{attribute 'global_init_slot' := '40510'}
VAR_GLOBAL
  LblFun_Requirement                                       :FB_BA_Label:=( sObjName:='REQ', sDescr:='Requirement');
  LblFun_SystemSwitch                                      :FB_BA_Label:=( sObjName:='PLS', sDescr:='Plant switch');
  LblFun_StatusOccupiedRoom                                :FB_BA_Label:=( sObjName:='OCC', sDescr:='Occupied status room');
  LblFun_LimitCalculatedValue                              :FB_BA_Label:=( sObjName:='LMC', sDescr:='Calculated limit value');
  LblFun_SetpointCalculated                                :FB_BA_Label:=( sObjName:='SPC', sDescr:='Calculated setpoint');
  LblFun_ReadyForOperation                                 :FB_BA_Label:=( sObjName:='RFO', sDescr:='Ready for operation');
  LblFun_OperationalMessage                                :FB_BA_Label:=( sObjName:='OM_', sDescr:='Operational message');
  LblFun_HoursOfOperation                                  :FB_BA_Label:=( sObjName:='OH_', sDescr:='Operating hours');
  LblFun_LimitValueHoursOfOperation                        :FB_BA_Label:=( sObjName:='OHL', sDescr:='Operating hours limit value');
  LblFun_ObjectCalendar                                    :FB_BA_Label:=( sObjName:='CAL', sDescr:='Calendar object');
  LblFun_ObjectCommand                                     :FB_BA_Label:=( sObjName:='COM', sDescr:='Command object');
  LblFun_DifferentialConstantController                    :FB_BA_Label:=( sObjName:='TV_', sDescr:='Differential constant controller');
  LblFun_SwitchOnErrorUnauthorisedON                       :FB_BA_Label:=( sObjName:='SWE', sDescr:='Switch-on error, unauthorised ON');
  LblFun_EnergyLevel                                       :FB_BA_Label:=( sObjName:='EL_', sDescr:='Energy level');
  LblFun_EnergyLevelCalculated                             :FB_BA_Label:=( sObjName:='ELC', sDescr:='Energy level calculated');
  LblFun_UnlockingDevice                                   :FB_BA_Label:=( sObjName:='UNL', sDescr:='Unlocking device');
  LblFun_ObjectEventEnrollment                             :FB_BA_Label:=( sObjName:='EE_', sDescr:='Event enrollment object');
  LblFun_Enabled                                           :FB_BA_Label:=( sObjName:='EN_', sDescr:='Enabled');
  LblFun_DangerAlarm                                       :FB_BA_Label:=( sObjName:='DA_', sDescr:='Danger alarm');
  LblFun_Threshold                                         :FB_BA_Label:=( sObjName:='LM_', sDescr:='Limit value');
  LblFun_LimitMAX                                          :FB_BA_Label:=( sObjName:='LMX', sDescr:='MAX limit');
  LblFun_LimitMIN                                          :FB_BA_Label:=( sObjName:='LMI', sDescr:='MIN limit');
  LblFun_LimitNight                                        :FB_BA_Label:=( sObjName:='LMN', sDescr:='Night limit');
  LblFun_LimitDay                                          :FB_BA_Label:=( sObjName:='LMD', sDescr:='Day limit');
  LblFun_ObjectGroup                                       :FB_BA_Label:=( sObjName:='GP_', sDescr:='Group object');
  LblFun_localPriorityAndOperatingUnitsManualMessage       :FB_BA_Label:=( sObjName:='MNM', sDescr:='local priority and operating units manual message');
  LblFun_HeatingCharacteristicCurveExponent                :FB_BA_Label:=( sObjName:='HEX', sDescr:='Heating characteristic curve exponent');
  LblFun_HeatingCharacteristicCurveParallelDisplacement    :FB_BA_Label:=( sObjName:='HPD', sDescr:='Heating characteristic curve parallel displacement');
  LblFun_HeatingCharacteristicCurveSteepness               :FB_BA_Label:=( sObjName:='HST', sDescr:='Heating characteristic curve steepness');
  LblFun_HeatingCircuitNightReduction                      :FB_BA_Label:=( sObjName:='NGT', sDescr:='Heating circuit night reduction');
  LblFun_Hysteresis                                        :FB_BA_Label:=( sObjName:='HYS', sDescr:='Hysteresis');
  LblFun_Calendar                                          :FB_BA_Label:=( sObjName:='CAL', sDescr:='Calendar');
  LblFun_RuntimeError                                      :FB_BA_Label:=( sObjName:='RUN', sDescr:='Runtime error');
  LblFun_LoopMAXLimit                                      :FB_BA_Label:=( sObjName:='LPX', sDescr:='Loop MAX limit');
  LblFun_LoopMINLimit                                      :FB_BA_Label:=( sObjName:='LPI', sDescr:='Loop MIN limit');
  LblFun_LoopObject                                        :FB_BA_Label:=( sObjName:='LP_', sDescr:='Loop object (controller object) – complex object');
  LblFun_LoopObjectCascadeSupplyAirTemperature             :FB_BA_Label:=( sObjName:='LP_', sDescr:='Cascade controller supply air temperature ');
  LblFun_LoopObjectCascadeSupplyAirHumidity                :FB_BA_Label:=( sObjName:='LP_', sDescr:='Cascade controller supply air humidity ');
  LblFun_MaximumValue                                      :FB_BA_Label:=( sObjName:='MAX', sDescr:='Maximum value');
  LblFun_MeasuredValue                                     :FB_BA_Label:=( sObjName:='MV_', sDescr:='Measured value');
  LblFun_MeasuredValueCalculated                           :FB_BA_Label:=( sObjName:='MVC', sDescr:='Measured value calculated');
  LblFun_MeasuredValueEast                                 :FB_BA_Label:=( sObjName:='MV_', sDescr:='Measured value East');
  LblFun_MeasuredValueNorth                                :FB_BA_Label:=( sObjName:='MV_', sDescr:='Measured value North');
  LblFun_MeasuredValueSouth                                :FB_BA_Label:=( sObjName:='MV_', sDescr:='Measured value South');
  LblFun_MeasuredValueWest                                 :FB_BA_Label:=( sObjName:='MV_', sDescr:='Measured value West');
  LblFun_MinimumValue                                      :FB_BA_Label:=( sObjName:='MIN', sDescr:='Minimum value');
  LblFun_Mean                                              :FB_BA_Label:=( sObjName:='MVL', sDescr:='Mean value');
  LblFun_FollowUpTime                                      :FB_BA_Label:=( sObjName:='FUT', sDescr:='Follow-up time');
  LblFun_ResetTime                                         :FB_BA_Label:=( sObjName:='RST', sDescr:='Reset time');
  LblFun_FeedbackDelay                                     :FB_BA_Label:=( sObjName:='TDF', sDescr:='Time delay feedback');
  LblFun_ObjectNotificationClass                           :FB_BA_Label:=( sObjName:='NC_', sDescr:='Notification class object');
  LblFun_EventClassObject                                  :FB_BA_Label:=( sObjName:='ECL', sDescr:='Event class');
  LblFun_Programobject                                     :FB_BA_Label:=( sObjName:='PRG', sDescr:='Program');
  LblFun_ProportionalBand                                  :FB_BA_Label:=( sObjName:='XP_', sDescr:='Proportional band');
  LblFun_FeedbackOPEN                                      :FB_BA_Label:=( sObjName:='FDO', sDescr:='Feedback OPEN');
  LblFun_FeedbackCLOSED                                    :FB_BA_Label:=( sObjName:='FDC', sDescr:='Feedback CLOSED');
  LblFun_FeedbackValue                                     :FB_BA_Label:=( sObjName:='FDB', sDescr:='Feedback value');
  LblFun_FeedbackErrorOPEN                                 :FB_BA_Label:=( sObjName:='FEO', sDescr:='Feedback error OPEN');
  LblFun_FeedbackErrorCLOSED                               :FB_BA_Label:=( sObjName:='FEC', sDescr:='Feedback error CLOSED');
  LblFun_Feedback                                          :FB_BA_Label:=( sObjName:='FDB', sDescr:='Feedback');
  LblFun_ExecutionControl                                  :FB_BA_Label:=( sObjName:='EXC', sDescr:='Execution control');
  LblFun_SwitchingCommand                                  :FB_BA_Label:=( sObjName:='SC_', sDescr:='Switching command');
  LblFun_Scheduler                                         :FB_BA_Label:=( sObjName:='SCH', sDescr:='Scheduler');
  LblFun_Setpoint                                          :FB_BA_Label:=( sObjName:='SP_', sDescr:='Setpoint');
  LblFun_SetpointComfortHeating                            :FB_BA_Label:=( sObjName:='SP_', sDescr:='Setpoint comfort heating');
  LblFun_SetpointPreComfortHeating                         :FB_BA_Label:=( sObjName:='SP_', sDescr:='Setpoint pre-comfort heating');
  LblFun_SetpointEconomyHeating                            :FB_BA_Label:=( sObjName:='SP_', sDescr:='Setpoint economy heating');
  LblFun_SetpointProtectionHeating                         :FB_BA_Label:=( sObjName:='SP_', sDescr:='Setpoint protection heating');
  LblFun_SetpointComfortCooling                            :FB_BA_Label:=( sObjName:='SP_', sDescr:='Setpoint comfort cooling');
  LblFun_SetpointPreComfortCooling                         :FB_BA_Label:=( sObjName:='SP_', sDescr:='Setpoint pre-comfort cooling');
  LblFun_SetpointEconomyCooling                            :FB_BA_Label:=( sObjName:='SP_', sDescr:='Setpoint economy cooling');
  LblFun_SetpointProtectionCooling                         :FB_BA_Label:=( sObjName:='SP_', sDescr:='Setpoint protection cooling');
  LblFun_SetpointBase                                      :FB_BA_Label:=( sObjName:='SPB', sDescr:='Base setpoint');
  LblFun_SetpointHeating                                   :FB_BA_Label:=( sObjName:='SPH', sDescr:='Heating setpoint');
  LblFun_SetpointCooling                                   :FB_BA_Label:=( sObjName:='SPC', sDescr:='Cooling setpoint');
  LblFun_SetpointMaximum                                   :FB_BA_Label:=( sObjName:='SPX', sDescr:='Setpoint, maximum');
  LblFun_SetpointMechanical                                :FB_BA_Label:=( sObjName:='SPM', sDescr:='Setpoint, mechanical');
  LblFun_SetpointMinimum                                   :FB_BA_Label:=( sObjName:='SPI', sDescr:='Setpoint, minimum');
  LblFun_SetpointNight                                     :FB_BA_Label:=( sObjName:='SPN', sDescr:='Night setpoint');
  LblFun_SetpointDay                                       :FB_BA_Label:=( sObjName:='SPD', sDescr:='Day setpoint');
  LblFun_SetpointAdjuster                                  :FB_BA_Label:=( sObjName:='SPA', sDescr:='Setpoint adjuster');
  LblFun_SetpointAdjustmentMechanical                      :FB_BA_Label:=( sObjName:='SPA', sDescr:='Setpoint adjustment, mechanical');
  LblFun_Selection                                         :FB_BA_Label:=( sObjName:='SEL', sDescr:='Selection');
  LblFun_Status                                            :FB_BA_Label:=( sObjName:='STA', sDescr:='Status');
  LblFun_ControlSignal                                     :FB_BA_Label:=( sObjName:='CS_', sDescr:='Control signal');
  LblFun_Fault                                             :FB_BA_Label:=( sObjName:='FAU', sDescr:='Fault');
  LblFun_FaultFuse                                         :FB_BA_Label:=( sObjName:='FAU', sDescr:='Fuse fault ');
  LblFun_Button                                            :FB_BA_Label:=( sObjName:='BUT', sDescr:='Button');
  LblFun_DeadZone                                          :FB_BA_Label:=( sObjName:='DZ_', sDescr:='Dead zone');
  LblFun_ObjectTrendLogMultiple                            :FB_BA_Label:=( sObjName:='TRM', sDescr:='Trend log multiple object');
  LblFun_ObjectTrendLog                                    :FB_BA_Label:=( sObjName:='TR_', sDescr:='Trend log object');
  LblFun_AmplificationController                           :FB_BA_Label:=( sObjName:='KP_', sDescr:='Amplification controller');
  LblFun_RetentionPeriod                                   :FB_BA_Label:=( sObjName:='TV_', sDescr:='Retention period');
  LblFun_MaintenanceMessage                                :FB_BA_Label:=( sObjName:='MTM', sDescr:='Maintenance message');
  LblFun_Efficiency                                        :FB_BA_Label:=( sObjName:='EFC', sDescr:='Efficiency');
  LblFun_CountValue                                        :FB_BA_Label:=( sObjName:='CNT', sDescr:='Count value');
  LblFun_TimeProgram                                       :FB_BA_Label:=( sObjName:='TPR', sDescr:='Time program');
//     Beckhoff Scale
  LblFun_ValueX1                                           :FB_BA_Label:=( sObjName:='IPX', sDescr:='Value interpolation point [X1]');
  LblFun_ValueX2                                           :FB_BA_Label:=( sObjName:='IPX', sDescr:='Value interpolation point [X2]');
  LblFun_ValueX3                                           :FB_BA_Label:=( sObjName:='IPX', sDescr:='Value interpolation point [X3]');
  LblFun_ValueX4                                           :FB_BA_Label:=( sObjName:='IPX', sDescr:='Value interpolation point [X4]');
  LblFun_ValueX5                                           :FB_BA_Label:=( sObjName:='IPX', sDescr:='Value interpolation point [X4]');
  LblFun_ValueX6                                           :FB_BA_Label:=( sObjName:='IPX', sDescr:='Value interpolation point [X4]');
  LblFun_ValueX7                                           :FB_BA_Label:=( sObjName:='IPX', sDescr:='Value interpolation point [X4]');
  LblFun_ValueY1                                           :FB_BA_Label:=( sObjName:='IPY', sDescr:='Value interpolation point [Y1]');
  LblFun_ValueY2                                           :FB_BA_Label:=( sObjName:='IPY', sDescr:='Value interpolation point [Y2]');
  LblFun_ValueY3                                           :FB_BA_Label:=( sObjName:='IPY', sDescr:='Value interpolation point [Y3]');
  LblFun_ValueY2_3                                         :FB_BA_Label:=( sObjName:='IPY', sDescr:='Value interpolation point [Y2-Y3]');
  LblFun_ValueY4                                           :FB_BA_Label:=( sObjName:='IPY', sDescr:='Value interpolation point [Y4]');
  LblFun_ValueY5                                           :FB_BA_Label:=( sObjName:='IPY', sDescr:='Value interpolation point [Y4]');
  LblFun_ValueY6                                           :FB_BA_Label:=( sObjName:='IPY', sDescr:='Value interpolation point [Y4]');
  LblFun_ValueY7                                           :FB_BA_Label:=( sObjName:='IPY', sDescr:='Value interpolation point [Y4]');
  LblFun_SuppyAirTempSetpointHeaterCalc                    :FB_BA_Label:=( sObjName:='SPC', sDescr:='Supply air Temperature setpoint heater calculated');
  LblFun_SuppyAirTempSetpointCoolerCalc                    :FB_BA_Label:=( sObjName:='SPC', sDescr:='Supply air Temperature setpoint cooler calculated');
  LblFun_SuppyAirTempSetpointERCCalc                       :FB_BA_Label:=( sObjName:='SPC', sDescr:='Supply air Temperature setpoint ERC calculated');
END_VAR

// ---- Templates/GVLs/Language/English/LblPlant_EN.TcGVL
{region '#Template'}
	{attribute 'Version' := '5.1.0.0'}
	{attribute 'Tags' := '"LCID": "1031", "Text": "GVL, DPAD, Plants, ObjectName, Description"'}
	{attribute 'Tags' := '"LCID": "1033", "Text": "GVL, DPAD, Plants, ObjectName, Description"'}
	{attribute 'Description' := '"LCID": "1031", "Text": "Textliste Anlagen"'}
	{attribute 'Description' := '"LCID": "1033", "Text": "Text list plants"'}
{endregion}

{attribute 'global_init_slot' := '40510'}
VAR_GLOBAL
  LblPlt_Facade                                            :FB_BA_Label:=( sObjName:='FAC',sDescr:='Facade');
  LblPlt_Natural_smoke_extraction                          :FB_BA_Label:=( sObjName:='NSE',sDescr:='Natural smoke extraction');
  LblPlt_Doors_gates_sluices                               :FB_BA_Label:=( sObjName:='DGS',sDescr:='Doors, gates, sluices');
  LblPlt_Smoke_and_heat_extraction_system                  :FB_BA_Label:=( sObjName:='SHV',sDescr:='Smoke and heat extraction system');
  LblPlt_Sunlight_protection                               :FB_BA_Label:=( sObjName:='SUN',sDescr:='Sunlight protection');
// 411 Sewage plants
  LblPlt_Separator_facility                                :FB_BA_Label:=( sObjName:='SEP',sDescr:='Separator facility');
  LblPlt_Lifting_system                                    :FB_BA_Label:=( sObjName:='LIF',sDescr:='Lifting system');
  LblPlt_Neutralisation_plant                              :FB_BA_Label:=( sObjName:='NEU',sDescr:='Neutralisation plant');
// 412 water plants
  LblPlt_Trace_heating                                     :FB_BA_Label:=( sObjName:='TRH',sDescr:='Trace heating');
  LblPlt_Process_water                                     :FB_BA_Label:=( sObjName:='PCW',sDescr:='Process water');
  LblPlt_Well_water                                        :FB_BA_Label:=( sObjName:='WWT',sDescr:='Well water');
  LblPlt_Dispensing_installation                           :FB_BA_Label:=( sObjName:='DPS',sDescr:='Dispensing installation');
  LblPlt_Pressure_booster_system                           :FB_BA_Label:=( sObjName:='PBS',sDescr:='Pressure booster system');
  LblPlt_Softening_unit                                    :FB_BA_Label:=( sObjName:='SOU',sDescr:='Softening unit');
// Drinking water
  LblPlt_Drinking_water_heating_system                     :FB_BA_Label:=( sObjName:='DWH',sDescr:='Drinking water heating system');
  LblPlt_Reverse_osmosis_system                            :FB_BA_Label:=( sObjName:='ROS',sDescr:='Reverse osmosis system');
  LblPlt_Desalination_plant                                :FB_BA_Label:=( sObjName:='SAP',sDescr:='Desalination plant');
// 421 Heat generation plants
  LblPlt_BHKW                                              :FB_BA_Label:=( sObjName:='BHK',sDescr:='BHKW');
  LblPlt_Electric_heating                                  :FB_BA_Label:=( sObjName:='EHT',sDescr:='Electric heating');
  LblPlt_District_heating_transfer                         :FB_BA_Label:=( sObjName:='DHT',sDescr:='District heating transfer');
// Geothermal system
  LblPlt_Boiler                                            :FB_BA_Label:=( sObjName:='BOI',sDescr:='Boiler');
  LblPlt_Clean_steam_generation                            :FB_BA_Label:=( sObjName:='CSG',sDescr:='Clean steam generation');
  LblPlt_Solar_power_system                                :FB_BA_Label:=( sObjName:='SOL',sDescr:='Solar power system');
  LblPlt_Heating_pump                                      :FB_BA_Label:=( sObjName:='HPU',sDescr:='Heating pump');
// 422 Heat distribution networks
  LblPlt_Pressure_maintenance                              :FB_BA_Label:=( sObjName:='PMT',sDescr:='Pressure maintenance');
  LblPlt_Heating_circuit                                   :FB_BA_Label:=( sObjName:='HTC',sDescr:='Heating circuit');
  LblPlt_Heating                                           :FB_BA_Label:=( sObjName:='HTG',sDescr:='Heating');
  LblPlt_Back_feed_system                                  :FB_BA_Label:=( sObjName:='BSF',sDescr:='Back-feed system');
  LblPlt_Buffer                                            :FB_BA_Label:=( sObjName:='BUF',sDescr:='Buffer');
  LblPlt_Heat_distribution_network                         :FB_BA_Label:=( sObjName:='HDN',sDescr:='Heat distribution network');
  LblPlt_Heat_exchanger                                    :FB_BA_Label:=( sObjName:='HEX',sDescr:='Heat exchanger');
// 423 Space-heating surfaces
  LblPlt_Concrete_core_activation                          :FB_BA_Label:=( sObjName:='CCA',sDescr:='Concrete core activation');
  LblPlt_Overhead_heating                                  :FB_BA_Label:=( sObjName:='OHH',sDescr:='Overhead heating');
  LblPlt_Ceiling_radiator_panels                           :FB_BA_Label:=( sObjName:='CRP',sDescr:='Ceiling radiator panels');
  LblPlt_Facade_heating                                    :FB_BA_Label:=( sObjName:='FAH',sDescr:='Facade heating');
  LblPlt_Panel_heating                                     :FB_BA_Label:=( sObjName:='PAH',sDescr:='Panel heating');
  LblPlt_Underfloor_heating                                :FB_BA_Label:=( sObjName:='UFH',sDescr:='Underfloor heating');
  LblPlt_Heated_chilled_ceiling                            :FB_BA_Label:=( sObjName:='HCC',sDescr:='Heated/chilled ceiling');
  LblPlt_Static_heating                                    :FB_BA_Label:=( sObjName:='STH',sDescr:='Static heating');
// 430 Ventilation systems
  LblPlt_Extract_air_system                                :FB_BA_Label:=( sObjName:='EXS',sDescr:='Extract air system');
  LblPlt_Roof_air_heater                                   :FB_BA_Label:=( sObjName:='RAH',sDescr:='Roof air heater');
  LblPlt_Circulatory_system                                :FB_BA_Label:=( sObjName:='CCS',sDescr:='Circulatory system');
  LblPlt_Air_processing_unit                               :FB_BA_Label:=( sObjName:='APU',sDescr:='Air processing unit');
  LblPlt_Mechanical_smoke_extraction_system                :FB_BA_Label:=( sObjName:='MSE',sDescr:='Mechanical smoke extraction system');
  LblPlt_Smoke_pressure_system                             :FB_BA_Label:=( sObjName:='SPS',sDescr:='Smoke pressure system');
  LblPlt_Air_handling_unit                                 :FB_BA_Label:=( sObjName:='AHU',sDescr:='Air handling unit');
  LblPlt_Partial_air_conditioning_system                   :FB_BA_Label:=( sObjName:='PAC',sDescr:='Partial air-conditioning system');
  LblPlt_Air_curtain_system                                :FB_BA_Label:=( sObjName:='ACS',sDescr:='Air curtain system');
  LblPlt_Recirculating_air_system                          :FB_BA_Label:=( sObjName:='RCA',sDescr:='Recirculating air system');
  LblPlt_Full_air_conditioning_system                      :FB_BA_Label:=( sObjName:='FAC',sDescr:='Full air-conditioning system');
  LblPlt_Heat_recovery_system                              :FB_BA_Label:=( sObjName:='REC',sDescr:='Heat recovery system');
  LblPlt_Intake_air_system                                 :FB_BA_Label:=( sObjName:='IAS',sDescr:='Intake air system');
  LblPlt_Smoke_extraction_system                           :FB_BA_Label:=( sObjName:='SME',sDescr:='Smoke extraction system');
// 434 Refrigeration systems
  LblPlt_Remote_cooling_transfer                           :FB_BA_Label:=( sObjName:='RCT',sDescr:='Remote cooling transfer');
  LblPlt_Cooling                                           :FB_BA_Label:=( sObjName:='COL',sDescr:='Cooling');
  LblPlt_Cooling_circuit                                   :FB_BA_Label:=( sObjName:='CCC',sDescr:='Cooling circuit');
  LblPlt_Cooling_distribution_network                      :FB_BA_Label:=( sObjName:='CDN',sDescr:='Cooling distribution network');
  LblPlt_Cold_water_generation                             :FB_BA_Label:=( sObjName:='CWG',sDescr:='Cold water generation');
  LblPlt_Electrical_cabinet_cooling                        :FB_BA_Label:=( sObjName:='ECC',sDescr:='Electrical cabinet cooling');
  LblPlt_Cooling_storage                                   :FB_BA_Label:=( sObjName:='CST',sDescr:='Cooling storage');
  LblPlt_Chilled_ceiling                                   :FB_BA_Label:=( sObjName:='CHC',sDescr:='Chilled ceiling');
  LblPlt_Re_cooling_plant                                  :FB_BA_Label:=( sObjName:='RCP',sDescr:='Re-cooling plant');
// 441 High and medium-voltage systems
  LblPlt_Switchgear                                        :FB_BA_Label:=( sObjName:='SWG',sDescr:='Switchgear');
  LblPlt_Transformer                                       :FB_BA_Label:=( sObjName:='TRF',sDescr:='Transformer');
  LblPlt_Medium_voltage_system                             :FB_BA_Label:=( sObjName:='MVS',sDescr:='Medium-voltage system');
  LblPlt_Compensation_system                               :FB_BA_Label:=( sObjName:='COS',sDescr:='Compensation system');
  LblPlt_Frequency_converter_system                        :FB_BA_Label:=( sObjName:='FCS',sDescr:='Frequency converter system');
// 442 Self-power supply systems
  LblPlt_Emissions_system                                  :FB_BA_Label:=( sObjName:='EMS',sDescr:='Emissions system');
  LblPlt_Battery_unit                                      :FB_BA_Label:=( sObjName:='BAT',sDescr:='Battery unit');
  LblPlt_Co_generation_unit                                :FB_BA_Label:=( sObjName:='CGU',sDescr:='Co-generation unit');
  LblPlt_Fuel_supply                                       :FB_BA_Label:=( sObjName:='FUS',sDescr:='Fuel supply');
  LblPlt_Standby_power_system                              :FB_BA_Label:=( sObjName:='SPS',sDescr:='Standby power system');
  LblPlt_Photovoltaic_system                               :FB_BA_Label:=( sObjName:='PVS',sDescr:='Photovoltaic system');
  LblPlt_Uninterruptible_power_supply                      :FB_BA_Label:=( sObjName:='UPS',sDescr:='Uninterruptible power supply');
// 443 Low-voltage switchgears
  LblPlt_General_power_supply                              :FB_BA_Label:=( sObjName:='GPS',sDescr:='General power supply');
  LblPlt_Safety_power_supply                               :FB_BA_Label:=( sObjName:='SPO',sDescr:='Safety power supply');
  LblPlt_Lighting                                          :FB_BA_Label:=( sObjName:='LIT',sDescr:='Lighting');
  LblPlt_Emergency_lighting                                :FB_BA_Label:=( sObjName:='EML',sDescr:='Emergency lighting');
// 451 Telecommunications systems
  LblPlt_Telecommunications_system                         :FB_BA_Label:=( sObjName:='TEL',sDescr:='Telecommunications system');
// 452 Search and signalling systems
  LblPlt_Call_signalling_system                            :FB_BA_Label:=( sObjName:='CSS',sDescr:='Call signalling system');
  LblPlt_Door_intercom_and_door_opener_system              :FB_BA_Label:=( sObjName:='DIO',sDescr:='Door intercom and door opener system');
  LblPlt_Paging_system                                     :FB_BA_Label:=( sObjName:='PGS',sDescr:='Paging system');
// 453 Time service systems
  LblPlt_Clock_and_time_recording_system                   :FB_BA_Label:=( sObjName:='CTR',sDescr:='Clock and time recording system');
// 454 Electro-acoustic systems
  LblPlt_Electro_acoustic_sound_systems                    :FB_BA_Label:=( sObjName:='ELA',sDescr:='Electro-acoustic system, sound systems');
  LblPlt_Conference_and_interpreting_equipment             :FB_BA_Label:=( sObjName:='CIE',sDescr:='Conference and interpreting equipment');
  LblPlt_Intercom_system                                   :FB_BA_Label:=( sObjName:='ICS',sDescr:='Intercom system');
  LblPlt_Voice_alarm_system                                :FB_BA_Label:=( sObjName:='VAS',sDescr:='Voice alarm system');
  LblPlt_Intercommunication_systems                        :FB_BA_Label:=( sObjName:='ICS',sDescr:='Intercommunication systems');
// 455 Television and antenna systems
  LblPlt_Television_system                                 :FB_BA_Label:=( sObjName:='TVS',sDescr:='Television system');
  LblPlt_Transmitting_and_receiving_antenna_system         :FB_BA_Label:=( sObjName:='TRA',sDescr:='Transmit. and receiving antenna system');
  LblPlt_BOS_radio_system                                  :FB_BA_Label:=( sObjName:='BOS',sDescr:='BOS radio system');
// 456 Hazard detection and alarm systems
  LblPlt_Fire_detection_and_alarm_systems                  :FB_BA_Label:=( sObjName:='FDA',sDescr:='Fire detection and alarm system');
  LblPlt_Carbon_monoxide_warning_system                    :FB_BA_Label:=( sObjName:='CMW',sDescr:='Carbon monoxide warning system');
  LblPlt_Burglar_alarm_systems                             :FB_BA_Label:=( sObjName:='BAS',sDescr:='Burglar alarm system');
  LblPlt_Fire_control_panel                                :FB_BA_Label:=( sObjName:='FCP',sDescr:='Fire control panel');
  LblPlt_Escape_route_protection_system                    :FB_BA_Label:=( sObjName:='ERP',sDescr:='Escape route protection system');
  LblPlt_Hazard_detection_system                           :FB_BA_Label:=( sObjName:='HDS',sDescr:='Hazard detection system');
  LblPlt_Gas_warning_system                                :FB_BA_Label:=( sObjName:='GWS',sDescr:='Gas warning system');
  LblPlt_Smoke_aspiration_system                           :FB_BA_Label:=( sObjName:='SAS',sDescr:='Smoke aspiration system');
  LblPlt_Room_observation_system                           :FB_BA_Label:=( sObjName:='ROS',sDescr:='Room observation system');
  LblPlt_Robbery_alarm_system                              :FB_BA_Label:=( sObjName:='ROA',sDescr:='Robbery alarm system');
  LblPlt_Guard_control_system                              :FB_BA_Label:=( sObjName:='GCS',sDescr:='Guard control system');
  LblPlt_Emergency_call_system                             :FB_BA_Label:=( sObjName:='EMG',sDescr:='Emergency call system');
  LblPlt_Access_control_system                             :FB_BA_Label:=( sObjName:='ACS',sDescr:='Access control system');
// 457 Transmission grids
  LblPlt_Networks_for_the_transmission_voice_text_etc      :FB_BA_Label:=( sObjName:='LAN',sDescr:='Networks  data, voice, text etc');
// 459 Telecommunication and information technology equipment, other
  LblPlt_Remote_control_systems                            :FB_BA_Label:=( sObjName:='RCS',sDescr:='Remote control systems');
  LblPlt_Parking_guidance_systems                          :FB_BA_Label:=( sObjName:='PGS',sDescr:='Parking guidance systems');
// 460 Conveyors
  LblPlt_File_transportation_systems                       :FB_BA_Label:=( sObjName:='FTS',sDescr:='File transportation systems');
  LblPlt_Lift                                              :FB_BA_Label:=( sObjName:='LIF',sDescr:='Lift');
  LblPlt_Inspection_systems                                :FB_BA_Label:=( sObjName:='ISS',sDescr:='Inspection systems');
  LblPlt_Moving_walkways                                   :FB_BA_Label:=( sObjName:='MWW',sDescr:='Moving walkways');
  LblPlt_Escalators                                        :FB_BA_Label:=( sObjName:='ESC',sDescr:='Escalators');
  LblPlt_External_lifts                                    :FB_BA_Label:=( sObjName:='EXL',sDescr:='External lifts');
  LblPlt_Baggage_conveyor_system                           :FB_BA_Label:=( sObjName:='BCS',sDescr:='Baggage conveyor system');
  LblPlt_Pneumatic_delivery_systems                        :FB_BA_Label:=( sObjName:='PDS',sDescr:='Pneumatic delivery systems');
  LblPlt_Goods_transportation_facilities                   :FB_BA_Label:=( sObjName:='GTF',sDescr:='Goods transportation facilities');
// 470 User-specific systems
// 471 Kitchen technology systems
  LblPlt_Small_refrigeration_unit                          :FB_BA_Label:=( sObjName:='SRU',sDescr:='Small refrigeration unit');
// 472 Laundry and cleaning systems
  LblPlt_Disinfection_unit                                 :FB_BA_Label:=( sObjName:='DIS',sDescr:='Disinfection unit');
  LblPlt_Cleaning_unit                                     :FB_BA_Label:=( sObjName:='CLU',sDescr:='Cleaning unit');
  LblPlt_Sterilisation_systems                             :FB_BA_Label:=( sObjName:='STR',sDescr:='Sterilisation systems');
  LblPlt_Water_treatment_system                            :FB_BA_Label:=( sObjName:='WTS',sDescr:='Water treatment system');
  LblPlt_Laundry_system                                    :FB_BA_Label:=( sObjName:='LAU',sDescr:='Laundry system');
// 473 Media supply systems
  LblPlt_Compressed_air_supply_system                      :FB_BA_Label:=( sObjName:='COA',sDescr:='Compressed air supply system');
  LblPlt_Pressure_regulator_unit                           :FB_BA_Label:=( sObjName:='PRU',sDescr:='Pressure regulator unit');
  LblPlt_Media_supply_system                               :FB_BA_Label:=( sObjName:='MSS',sDescr:='Media supply system');
  LblPlt_Medical_and_technical_gases                       :FB_BA_Label:=( sObjName:='MTG',sDescr:='Medical and technical gases');
  LblPlt_Vacuum_unit                                       :FB_BA_Label:=( sObjName:='VAC',sDescr:='Vacuum unit');
// 474 Medical and laboratory equipment
  LblPlt_Medical_technical_plant                           :FB_BA_Label:=( sObjName:='MED',sDescr:='Medical technical plant');
  LblPlt_Medical_gas_supply                                :FB_BA_Label:=( sObjName:='MGS',sDescr:='Medical gas supply');
  LblPlt_Laboratory_equipment                              :FB_BA_Label:=( sObjName:='LAB',sDescr:='Laboratory equipment (general)');
// 475 Fire extinguishers
  LblPlt_Fire_extinguisher                                 :FB_BA_Label:=( sObjName:='FEG',sDescr:='Fire extinguisher');
  LblPlt_Gas_extinguishing_system                          :FB_BA_Label:=( sObjName:='GES',sDescr:='Gas extinguishing system');
  LblPlt_Fire_extinguishing_system                         :FB_BA_Label:=( sObjName:='FES',sDescr:='Fire extinguishing system (general)');
  LblPlt_Mist_extinguishing_system                         :FB_BA_Label:=( sObjName:='MES',sDescr:='Mist-extinguishing system');
  LblPlt_NOX_system                                        :FB_BA_Label:=( sObjName:='NOX',sDescr:='NOX system');
  LblPlt_Sprinkler_system                                  :FB_BA_Label:=( sObjName:='SPR',sDescr:='Sprinkler system');
  LblPlt_Wall_hydrant_system                               :FB_BA_Label:=( sObjName:='WHS',sDescr:='Wall hydrant system');
// 478 Disposal facilities
  LblPlt_Waste_disposal_system                             :FB_BA_Label:=( sObjName:='WDS',sDescr:='Waste disposal system');
  LblPlt_Media_disposal_system                             :FB_BA_Label:=( sObjName:='MDS',sDescr:='Media disposal system');
  LblPlt_Vacuum_cleaning_systems                           :FB_BA_Label:=( sObjName:='VCS',sDescr:='Vacuum cleaning systems');
// 480 Building automation and control systems
  LblPlt_Automation_control_equipment                      :FB_BA_Label:=( sObjName:='ACE',sDescr:='Automation and control equipment');
  LblPlt_Weather_station                                   :FB_BA_Label:=( sObjName:='WET',sDescr:='Weather station');
  LblPlt_Weather_data                                      :FB_BA_Label:=( sObjName:='WED',sDescr:='Weather data');
  LblPlt_Management_and_operating_equipment                :FB_BA_Label:=( sObjName:='MOE',sDescr:='Management and operating equipment');
  LblPlt_Room_automation                                   :FB_BA_Label:=( sObjName:='RAU',sDescr:='Room automation');
  LblPlt_Room_automation_system_distributor                :FB_BA_Label:=( sObjName:='RAS',sDescr:='Room automation system distributor');
  LblPlt_Control_cabinet                                   :FB_BA_Label:=( sObjName:='CCB',sDescr:='Control cabinet');
  LblPlt_Settings                                          :FB_BA_Label:=( sObjName:='SYP',sDescr:='System parameters');
  LblPlt_EventGroups                                       :FB_BA_Label:=( sObjName:='EVG',sDescr:='Event groups');
  LblPlt_Global_building_data                              :FB_BA_Label:=( sObjName:='GBD',sDescr:='Global building data');
// 540 Technical equipment in outdoor facilities
  LblPlt_Rainwater_retention_basin                         :FB_BA_Label:=( sObjName:='RRB',sDescr:='Rainwater retention basin');
  LblPlt_Cistern_system                                    :FB_BA_Label:=( sObjName:='CIS',sDescr:='Cistern system');
END_VAR

// ---- Templates/GVLs/Language/English/TxtEvent_EN.TcGVL
{region '#Template'}
	{attribute 'Version' := '5.1.0.0'}
	{attribute 'Tags' := '"LCID": "1031", "Text": "GVL, Property, Event, Event Message Text, Active Text, Inactive Text"'}
	{attribute 'Tags' := '"LCID": "1033", "Text": "GVL, Property, Event, Event Message Text, Active Text, Inactive Text"'}
	{attribute 'Description' := '"LCID": "1031", "Text": "Textliste Properties Event Message Text, Active Text, Inactive Text"'}
	{attribute 'Description' := '"LCID": "1033", "Text": "Text list Properties Event Message Text, Active Text, Inactive Text"'}
{endregion}

{attribute 'global_init_slot' := '40510'}
VAR_GLOBAL
  txtEvent_No                                                :T_BA_StateText:='No';
  txtEvent_Yes                                               :T_BA_StateText:='Yes';
  txtEvent_Auto                                              :T_BA_StateText:='Auto';
  txtEvent_Manual                                            :T_BA_StateText:='Manual';
  txtEvent_Off                                               :T_BA_StateText:='Off';
  txtEvent_On                                                :T_BA_StateText:='On';
  txtEvent_Opened                                            :T_BA_StateText:='Opened';
  txtEvent_Closed                                            :T_BA_StateText:='Closed';
  txtEvent_Open                                              :T_BA_StateText:='Open';
  txtEvent_Close                                             :T_BA_StateText:='Close';
  txtEvent_Step1                                             :T_BA_StateText:='Step1';
  txtEvent_Step2                                             :T_BA_StateText:='Step2';
  txtEvent_Step3                                             :T_BA_StateText:='Step3';
  txtEvent_Step4                                             :T_BA_StateText:='Step4';
  txtEvent_Step5                                             :T_BA_StateText:='Step5';
  txtEvent_Step6                                             :T_BA_StateText:='Step6';
  txtEvent_Step7                                             :T_BA_StateText:='Step7';
  txtEvent_Step8                                             :T_BA_StateText:='Step8';
  txtEvent_Released                                          :T_BA_StateText:='Released';
  txtEvent_Inactive                                          :T_BA_StateText:='Inactive';
  txtEvent_Active                                            :T_BA_StateText:='Active';
  txtEvent_Normal                                            :T_BA_StateText:='Normal';
  txtEvent_Offnormal                                         :T_BA_StateText:='Offnormal';
  txtEvent_Alert                                             :T_BA_StateText:='Alert';
  txtEvent_Disturb                                           :T_BA_StateText:='Disturb';
  txtEvent_Error                                             :T_BA_StateText:='Error';
  txtEvent_Triggered                                         :T_BA_StateText:='Triggered';
  txtEvent_Maintenace                                        :T_BA_StateText:='Maintenace';
  txtEvent_Exceeded                                          :T_BA_StateText:='Exceeded';
  txtEvent_Monitoring                                        :T_BA_StateText:='Monitoring';
  txtEvent_Protection                                        :T_BA_StateText:='Protection';
  txtEvent_Economy                                           :T_BA_StateText:='Economy';
  txtEvent_PreComfort                                        :T_BA_StateText:='PreComfort';
  txtEvent_Comfort                                           :T_BA_StateText:='Comfort';
  txtEvent_Reached                                           :T_BA_StateText:='Reached';
  txtEvent_NotReached                                        :T_BA_StateText:='NotReached';
  txtEvent_None                                              :T_BA_StateText:='None';
  txtEvent_EmergencyStop                                     :T_BA_StateText:='EmergencyStop';
  txtEvent_Frost                                             :T_BA_StateText:='Frost';
  txtEvent_SmokeExtraction_P                                 :T_BA_StateText:='SmokeExtraction_P';
  txtEvent_SmokeExtractionSupplyAir                          :T_BA_StateText:='SmokeExtractionSupplyAir';
  txtEvent_SmokeExtractionExtractAir                         :T_BA_StateText:='SmokeExtractionExtractAir';
  txtEvent_CoolDownProtection                                :T_BA_StateText:='CoolDownProtection';
  txtEvent_OverHeatingProtection                             :T_BA_StateText:='OverHeatingProtection';
  txtEvent_Fire                                              :T_BA_StateText:='Fire';
  txtEvent_NightCooling                                      :T_BA_StateText:='NightCooling';
  txtEvent_ForcedVentilation                                 :T_BA_StateText:='ForcedVentilation';
  txtEvent_CentralSwitchOff                                  :T_BA_StateText:='CentralSwitchOff';
  txtEvent_Locked                                            :T_BA_StateText:='Locked';
  txtEvent_Contaminated                                      :T_BA_StateText:='Contaminated';
  txtEvent_Stop                                              :T_BA_StateText:='Stop';
  txtEvent_Critical                                          :T_BA_StateText:='Critical';
  txtEvent_CriticalOn                                        :T_BA_StateText:='Critical on';
  txtEvent_CriticalOff                                       :T_BA_StateText:='Critical off';
  txtEvent_UnCiritical                                       :T_BA_StateText:='UnCiritical';
  txtEvent_LifeSafetyOn                                      :T_BA_StateText:='Life safety on';
  txtEvent_LifeSafetyOff                                     :T_BA_StateText:='Life safety off';
  txtEvent_Average                                           :T_BA_StateText:='Average';
  txtEvent_HeatCool                                          :T_BA_StateText:='HeatCool';
  txtEvent_AverageHeatCool                                   :T_BA_StateText:='AverageHeatCool';
  txtEvent_Direction                                         :T_BA_StateText:='Direction';
  txtEvent_Default                                           :T_BA_StateText:='Default';
  txtEvent_Cleaning                                          :T_BA_StateText:='Cleaning';
  txtEvent_Nightwatch                                        :T_BA_StateText:='Nightwatch';
  txtEvent_SupplyAirTControlReheater                         :T_BA_StateText:='Supply air temp control reheater';
  txtEvent_SupplyAirTControlPreheater                        :T_BA_StateText:='Supply air temp control preheater';
  txtEvent_SupplyAirTControlERC                              :T_BA_StateText:='Supply air temp control ERC';
  txtEvent_SupplyAirTControlMix                              :T_BA_StateText:='Supply air temp control mixed air';
  txtEvent_SupplyAirTControlCooler                           :T_BA_StateText:='Supply air temp control cooler';
  txtEvent_SupplyAirXControlCooler                           :T_BA_StateText:='Supply air humidity control cooler';
  txtEvent_SupplyAirXControlHumf                             :T_BA_StateText:='Supply air humidity control humidifier';
  txtEvent_PreRinse                                          :T_BA_StateText:='Pre Rinse';
  txtEvent_DamperOpen                                        :T_BA_StateText:='Damper Open';
  txtEvent_SupplyAirFan                                      :T_BA_StateText:='Supply Air Fan';
  txtEvent_ExtractAirFan                                     :T_BA_StateText:='Extract Air Fan';
  txtEvent_EnableTemperatureControl                          :T_BA_StateText:='Enable Temperature Control';
  txtEvent_EnableTemperatureSequenceLink                     :T_BA_StateText:='Enable Temperature Sequence Link';
  txtEvent_EnableHumidityControl                             :T_BA_StateText:='Enable Humidity Control';
  txtEvent_EnableHumiditySequenceLink                        :T_BA_StateText:='Enable Humidity Sequence Link';
  txtEvent_ReleaseLimitMonitoring                            :T_BA_StateText:='Release Limit Monitoring';
  txtEvent_Reheater                                          :T_BA_StateText:='Reheater';
  txtEvent_Preheater                                         :T_BA_StateText:='Preheater';
  txtEvent_MixedAir                                          :T_BA_StateText:='Mixed Air';
  txtEvent_EnergyRecovery                                    :T_BA_StateText:='Energy Recovery';
  txtEvent_Cooler                                            :T_BA_StateText:='Cooler';
  txtEvent_Humidifier                                        :T_BA_StateText:='Humidifier';
  txtEvent_Dehumidifier                                      :T_BA_StateText:='Dehumidifier';
  txtEvent_DamperExhaustAir                                  :T_BA_StateText:='Damper exhaust air';
  txtEvent_DamperOutsideAir                                  :T_BA_StateText:='Damper outside air';
  txtEvent_Occupied                                          :T_BA_StateText:='Occupied';
  txtEvent_NotOccupied                                       :T_BA_StateText:='Not occupied';
  txtEvent_Storm                                             :T_BA_StateText:='Storm-alarm';
  txtEvent_Ice                                               :T_BA_StateText:='Ice-alarm';
  txtEvent_CommError                                         :T_BA_StateText:='Communication-error';
  txtEvent_Burglary                                          :T_BA_StateText:='Burglary';
  txtEvent_Maintenance                                       :T_BA_StateText:='Maintenance';
  txtEvent_Referencing                                       :T_BA_StateText:='Referencing';
  txtEvent_ManualActuator                                    :T_BA_StateText:='Manual actuator';
  txtEvent_ManualGroup                                       :T_BA_StateText:='Manual group';
  txtEvent_AllDown                                           :T_BA_StateText:='All down';
  txtEvent_AllUp                                             :T_BA_StateText:='All up';
  txtEvent_Scene1                                            :T_BA_StateText:='Scene 1';
  txtEvent_FacadeThermoAutomatic                             :T_BA_StateText:='Facade thermo automatic';
  txtEvent_FacadeTwilightAutomatic                           :T_BA_StateText:='Facade twilight automatic';
  txtEvent_ParkPosition                                      :T_BA_StateText:='Park position';
  txtEvent_Scene2                                            :T_BA_StateText:='Scene2';
  txtEvent_Scene3                                            :T_BA_StateText:='Scene3';
  txtEvent_SunProtection                                     :T_BA_StateText:='Sun protection';
  txtEvent_GroupThermoAuto                                   :T_BA_StateText:='Group thermo automatic';
  txtEvent_GroupTwiLightAuto                                 :T_BA_StateText:='Group twilight automatic';
  txtEvent_UserDefined1                                      :T_BA_StateText:='Userdefined 1';
  txtEvent_UserDefined2                                      :T_BA_StateText:='Userdefined 2';
END_VAR

// ---- Templates/GVLs/Language/English/TxtPlant_EN.TcGVL
{region '#Template'}
	{attribute 'Version' := '5.0.2.0'}
	{attribute 'Tags' := '"LCID": "1031", "Text": "GVL, DPAD, Plants, ObjectName, Description"'}
	{attribute 'Tags' := '"LCID": "1033", "Text": "GVL, DPAD, Plants, ObjectName, Description"'}
	{attribute 'Description' := '"LCID": "1031", "Text": "Textliste Anlagen"'}
	{attribute 'Description' := '"LCID": "1033", "Text": "Text list plants"'}
{endregion}

{attribute 'global_init_slot' := '40510'}
VAR_GLOBAL
  TxTPlant_Facade_sObjectName                                            :T_BA_StateText:='FAC';
  TxTPlant_Facade_sDescription                                            :T_BA_StateText:='Facade';
  TxTPlant_Natural_smoke_extraction_sObjectName                          :T_BA_StateText:='NSE';
  TxTPlant_Natural_smoke_extraction_sDescription                          :T_BA_StateText:='Natural smoke extraction';
  TxTPlant_Doors_gates_sluices_sObjectName                               :T_BA_StateText:='DGS';
  TxTPlant_Doors_gates_sluices_sDescription                               :T_BA_StateText:='Doors, gates, sluices';
  TxTPlant_Smoke_and_heat_extraction_system_sObjectName                  :T_BA_StateText:='SHV';
  TxTPlant_Smoke_and_heat_extraction_system_sDescription                  :T_BA_StateText:='Smoke and heat extraction system';
  TxTPlant_Sunlight_protection_sObjectName                               :T_BA_StateText:='SUN';
  TxTPlant_Sunlight_protection_sDescription                               :T_BA_StateText:='Sunlight protection';
// 411 Sewage plants
  TxTPlant_Separator_facility_sObjectName                                :T_BA_StateText:='SEP';
  TxTPlant_Separator_facility_sDescription                                :T_BA_StateText:='Separator facility';
  TxTPlant_Lifting_system_sObjectName                                    :T_BA_StateText:='LIF';
  TxTPlant_Lifting_system_sDescription                                    :T_BA_StateText:='Lifting system';
  TxTPlant_Neutralisation_plant_sObjectName                              :T_BA_StateText:='NEU';
  TxTPlant_Neutralisation_plant_sDescription                              :T_BA_StateText:='Neutralisation plant';
// 412 water plants
  TxTPlant_Trace_heating_sObjectName                                     :T_BA_StateText:='TRH';
  TxTPlant_Trace_heating_sDescription                                     :T_BA_StateText:='Trace heating';
  TxTPlant_Process_water_sObjectName                                     :T_BA_StateText:='PCW';
  TxTPlant_Process_water_sDescription                                     :T_BA_StateText:='Process water';
  TxTPlant_Well_water_sObjectName                                        :T_BA_StateText:='WWT';
  TxTPlant_Well_water_sDescription                                        :T_BA_StateText:='Well water';
  TxTPlant_Dispensing_installation_sObjectName                           :T_BA_StateText:='DPS';
  TxTPlant_Dispensing_installation_sDescription                           :T_BA_StateText:='Dispensing installation';
  TxTPlant_Pressure_booster_system_sObjectName                           :T_BA_StateText:='PBS';
  TxTPlant_Pressure_booster_system_sDescription                           :T_BA_StateText:='Pressure booster system';
  TxTPlant_Softening_unit_sObjectName                                    :T_BA_StateText:='SOU';
  TxTPlant_Softening_unit_sDescription                                    :T_BA_StateText:='Softening unit';
// Drinking water
  TxTPlant_Drinking_water_heating_system_sObjectName                     :T_BA_StateText:='DWH';
  TxTPlant_Drinking_water_heating_system_sDescription                     :T_BA_StateText:='Drinking water heating system';
  TxTPlant_Reverse_osmosis_system_sObjectName                            :T_BA_StateText:='ROS';
  TxTPlant_Reverse_osmosis_system_sDescription                            :T_BA_StateText:='Reverse osmosis system';
  TxTPlant_Desalination_plant_sObjectName                                :T_BA_StateText:='SAP';
  TxTPlant_Desalination_plant_sDescription                                :T_BA_StateText:='Desalination plant';
// 421 Heat generation plants
  TxTPlant_BHKW_sObjectName                                              :T_BA_StateText:='BHK';
  TxTPlant_BHKW_sDescription                                              :T_BA_StateText:='BHKW';
  TxTPlant_Electric_heating_sObjectName                                  :T_BA_StateText:='EHT';
  TxTPlant_Electric_heating_sDescription                                  :T_BA_StateText:='Electric heating';
  TxTPlant_District_heating_transfer_sObjectName                         :T_BA_StateText:='DHT';
  TxTPlant_District_heating_transfer_sDescription                         :T_BA_StateText:='District heating transfer';
// Geothermal system
  TxTPlant_Boiler_sObjectName                                            :T_BA_StateText:='BOI';
  TxTPlant_Boiler_sDescription                                            :T_BA_StateText:='Boiler';
  TxTPlant_Clean_steam_generation_sObjectName                            :T_BA_StateText:='CSG';
  TxTPlant_Clean_steam_generation_sDescription                            :T_BA_StateText:='Clean steam generation';
  TxTPlant_Solar_power_system_sObjectName                                :T_BA_StateText:='SOL';
  TxTPlant_Solar_power_system_sDescription                                :T_BA_StateText:='Solar power system';
  TxTPlant_Heating_pump_sObjectName                                      :T_BA_StateText:='HPU';
  TxTPlant_Heating_pump_sDescription                                      :T_BA_StateText:='Heating pump';
// 422 Heat distribution networks
  TxTPlant_Pressure_maintenance_sObjectName                              :T_BA_StateText:='PMT';
  TxTPlant_Pressure_maintenance_sDescription                              :T_BA_StateText:='Pressure maintenance';
  TxTPlant_Heating_circuit_sObjectName                                   :T_BA_StateText:='HTC';
  TxTPlant_Heating_circuit_sDescription                                   :T_BA_StateText:='Heating circuit';
  TxTPlant_Heating_sObjectName                                           :T_BA_StateText:='HTG';
  TxTPlant_Heating_sDescription                                           :T_BA_StateText:='Heating';
  TxTPlant_Back_feed_system_sObjectName                                  :T_BA_StateText:='BSF';
  TxTPlant_Back_feed_system_sDescription                                  :T_BA_StateText:='Back-feed system';
  TxTPlant_Buffer_sObjectName                                            :T_BA_StateText:='BUF';
  TxTPlant_Buffer_sDescription                                            :T_BA_StateText:='Buffer';
  TxTPlant_Heat_distribution_network_sObjectName                         :T_BA_StateText:='HDN';
  TxTPlant_Heat_distribution_network_sDescription                         :T_BA_StateText:='Heat distribution network';
  TxTPlant_Heat_exchanger_sObjectName                                    :T_BA_StateText:='HEX';
  TxTPlant_Heat_exchanger_sDescription                                    :T_BA_StateText:='Heat exchanger';
// 423 Space-heating surfaces
  TxTPlant_Concrete_core_activation_sObjectName                          :T_BA_StateText:='CCA';
  TxTPlant_Concrete_core_activation_sDescription                          :T_BA_StateText:='Concrete core activation';
  TxTPlant_Overhead_heating_sObjectName                                  :T_BA_StateText:='OHH';
  TxTPlant_Overhead_heating_sDescription                                  :T_BA_StateText:='Overhead heating';
  TxTPlant_Ceiling_radiator_panels_sObjectName                           :T_BA_StateText:='CRP';
  TxTPlant_Ceiling_radiator_panels_sDescription                           :T_BA_StateText:='Ceiling radiator panels';
  TxTPlant_Facade_heating_sObjectName                                    :T_BA_StateText:='FAH';
  TxTPlant_Facade_heating_sDescription                                    :T_BA_StateText:='Facade heating';
  TxTPlant_Panel_heating_sObjectName                                     :T_BA_StateText:='PAH';
  TxTPlant_Panel_heating_sDescription                                     :T_BA_StateText:='Panel heating';
  TxTPlant_Underfloor_heating_sObjectName                                :T_BA_StateText:='UFH';
  TxTPlant_Underfloor_heating_sDescription                                :T_BA_StateText:='Underfloor heating';
  TxTPlant_Heated_chilled_ceiling_sObjectName                            :T_BA_StateText:='HCC';
  TxTPlant_Heated_chilled_ceiling_sDescription                            :T_BA_StateText:='Heated/chilled ceiling';
  TxTPlant_Static_heating_sObjectName                                    :T_BA_StateText:='STH';
  TxTPlant_Static_heating_sDescription                                    :T_BA_StateText:='Static heating';
// 430 Ventilation systems
  TxTPlant_Extract_air_system_sObjectName                                :T_BA_StateText:='EXS';
  TxTPlant_Extract_air_system_sDescription                                :T_BA_StateText:='Extract air system';
  TxTPlant_Roof_air_heater_sObjectName                                   :T_BA_StateText:='RAH';
  TxTPlant_Roof_air_heater_sDescription                                   :T_BA_StateText:='Roof air heater';
  TxTPlant_Circulatory_system_sObjectName                                :T_BA_StateText:='CCS';
  TxTPlant_Circulatory_system_sDescription                                :T_BA_StateText:='Circulatory system';
  TxTPlant_Air_processing_unit_sObjectName                               :T_BA_StateText:='APU';
  TxTPlant_Air_processing_unit_sDescription                               :T_BA_StateText:='Air processing unit';
  TxTPlant_Mechanical_smoke_extraction_system_sObjectName                :T_BA_StateText:='MSE';
  TxTPlant_Mechanical_smoke_extraction_system_sDescription                :T_BA_StateText:='Mechanical smoke extraction system';
  TxTPlant_Smoke_pressure_system_sObjectName                             :T_BA_StateText:='SPS';
  TxTPlant_Smoke_pressure_system_sDescription                             :T_BA_StateText:='Smoke pressure system';
  TxTPlant_Air_handling_unit_sObjectName                                 :T_BA_StateText:='AHU';
  TxTPlant_Air_handling_unit_sDescription                                 :T_BA_StateText:='Air handling unit';
  TxTPlant_Partial_air_conditioning_system_sObjectName                   :T_BA_StateText:='PAC';
  TxTPlant_Partial_air_conditioning_system_sDescription                   :T_BA_StateText:='Partial air-conditioning system';
  TxTPlant_Air_curtain_system_sObjectName                                :T_BA_StateText:='ACS';
  TxTPlant_Air_curtain_system_sDescription                                :T_BA_StateText:='Air curtain system';
  TxTPlant_Recirculating_air_system_sObjectName                          :T_BA_StateText:='RCA';
  TxTPlant_Recirculating_air_system_sDescription                          :T_BA_StateText:='Recirculating air system';
  TxTPlant_Full_air_conditioning_system_sObjectName                      :T_BA_StateText:='FAC';
  TxTPlant_Full_air_conditioning_system_sDescription                      :T_BA_StateText:='Full air-conditioning system';
  TxTPlant_Heat_recovery_system_sObjectName                              :T_BA_StateText:='REC';
  TxTPlant_Heat_recovery_system_sDescription                              :T_BA_StateText:='Heat recovery system';
  TxTPlant_Intake_air_system_sObjectName                                 :T_BA_StateText:='IAS';
  TxTPlant_Intake_air_system_sDescription                                 :T_BA_StateText:='Intake air system';
  TxTPlant_Smoke_extraction_system_sObjectName                           :T_BA_StateText:='SME';
  TxTPlant_Smoke_extraction_system_sDescription                           :T_BA_StateText:='Smoke extraction system';
// 434 Refrigeration systems
  TxTPlant_Remote_cooling_transfer_sObjectName                           :T_BA_StateText:='RCT';
  TxTPlant_Remote_cooling_transfer_sDescription                           :T_BA_StateText:='Remote cooling transfer';
  TxTPlant_Cooling_sObjectName                                           :T_BA_StateText:='COL';
  TxTPlant_Cooling_sDescription                                           :T_BA_StateText:='Cooling';
  TxTPlant_Cooling_circuit_sObjectName                                   :T_BA_StateText:='CCC';
  TxTPlant_Cooling_circuit_sDescription                                   :T_BA_StateText:='Cooling circuit';
  TxTPlant_Cooling_distribution_network_sObjectName                      :T_BA_StateText:='CDN';
  TxTPlant_Cooling_distribution_network_sDescription                      :T_BA_StateText:='Cooling distribution network';
  TxTPlant_Cold_water_generation_sObjectName                             :T_BA_StateText:='CWG';
  TxTPlant_Cold_water_generation_sDescription                             :T_BA_StateText:='Cold water generation';
  TxTPlant_Electrical_cabinet_cooling_sObjectName                        :T_BA_StateText:='ECC';
  TxTPlant_Electrical_cabinet_cooling_sDescription                        :T_BA_StateText:='Electrical cabinet cooling';
  TxTPlant_Cooling_storage_sObjectName                                   :T_BA_StateText:='CST';
  TxTPlant_Cooling_storage_sDescription                                   :T_BA_StateText:='Cooling storage';
  TxTPlant_Chilled_ceiling_sObjectName                                   :T_BA_StateText:='CHC';
  TxTPlant_Chilled_ceiling_sDescription                                   :T_BA_StateText:='Chilled ceiling';
  TxTPlant_Re_cooling_plant_sObjectName                                  :T_BA_StateText:='RCP';
  TxTPlant_Re_cooling_plant_sDescription                                  :T_BA_StateText:='Re-cooling plant';
// 441 High and medium-voltage systems
  TxTPlant_Switchgear_sObjectName                                        :T_BA_StateText:='SWG';
  TxTPlant_Switchgear_sDescription                                        :T_BA_StateText:='Switchgear';
  TxTPlant_Transformer_sObjectName                                       :T_BA_StateText:='TRF';
  TxTPlant_Transformer_sDescription                                       :T_BA_StateText:='Transformer';
  TxTPlant_Medium_voltage_system_sObjectName                             :T_BA_StateText:='MVS';
  TxTPlant_Medium_voltage_system_sDescription                             :T_BA_StateText:='Medium-voltage system';
  TxTPlant_Compensation_system_sObjectName                               :T_BA_StateText:='COS';
  TxTPlant_Compensation_system_sDescription                               :T_BA_StateText:='Compensation system';
  TxTPlant_Frequency_converter_system_sObjectName                        :T_BA_StateText:='FCS';
  TxTPlant_Frequency_converter_system_sDescription                        :T_BA_StateText:='Frequency converter system';
// 442 Self-power supply systems
  TxTPlant_Emissions_system_sObjectName                                  :T_BA_StateText:='EMS';
  TxTPlant_Emissions_system_sDescription                                  :T_BA_StateText:='Emissions system';
  TxTPlant_Battery_unit_sObjectName                                      :T_BA_StateText:='BAT';
  TxTPlant_Battery_unit_sDescription                                      :T_BA_StateText:='Battery unit';
  TxTPlant_Co_generation_unit_sObjectName                                :T_BA_StateText:='CGU';
  TxTPlant_Co_generation_unit_sDescription                                :T_BA_StateText:='Co-generation unit';
  TxTPlant_Fuel_supply_sObjectName                                       :T_BA_StateText:='FUS';
  TxTPlant_Fuel_supply_sDescription                                       :T_BA_StateText:='Fuel supply';
  TxTPlant_Standby_power_system_sObjectName                              :T_BA_StateText:='SPS';
  TxTPlant_Standby_power_system_sDescription                              :T_BA_StateText:='Standby power system';
  TxTPlant_Photovoltaic_system_sObjectName                               :T_BA_StateText:='PVS';
  TxTPlant_Photovoltaic_system_sDescription                               :T_BA_StateText:='Photovoltaic system';
  TxTPlant_Uninterruptible_power_supply_sObjectName                      :T_BA_StateText:='UPS';
  TxTPlant_Uninterruptible_power_supply_sDescription                      :T_BA_StateText:='Uninterruptible power supply';
// 443 Low-voltage switchgears
  TxTPlant_General_power_supply_sObjectName                              :T_BA_StateText:='GPS';
  TxTPlant_General_power_supply_sDescription                              :T_BA_StateText:='General power supply';
  TxTPlant_Safety_power_supply_sObjectName                               :T_BA_StateText:='SPO';
  TxTPlant_Safety_power_supply_sDescription                               :T_BA_StateText:='Safety power supply';
  TxTPlant_Lighting_sObjectName                                          :T_BA_StateText:='LIT';
  TxTPlant_Lighting_sDescription                                          :T_BA_StateText:='Lighting';
  TxTPlant_Emergency_lighting_sObjectName                                :T_BA_StateText:='EML';
  TxTPlant_Emergency_lighting_sDescription                                :T_BA_StateText:='Emergency lighting';
// 451 Telecommunications systems
  TxTPlant_Telecommunications_system_sObjectName                         :T_BA_StateText:='TEL';
  TxTPlant_Telecommunications_system_sDescription                         :T_BA_StateText:='Telecommunications system';
// 452 Search and signalling systems
  TxTPlant_Call_signalling_system_sObjectName                            :T_BA_StateText:='CSS';
  TxTPlant_Call_signalling_system_sDescription                            :T_BA_StateText:='Call signalling system';
  TxTPlant_Door_intercom_and_door_opener_system_sObjectName              :T_BA_StateText:='DIO';
  TxTPlant_Door_intercom_and_door_opener_system_sDescription              :T_BA_StateText:='Door intercom and door opener system';
  TxTPlant_Paging_system_sObjectName                                     :T_BA_StateText:='PGS';
  TxTPlant_Paging_system_sDescription                                     :T_BA_StateText:='Paging system';
// 453 Time service systems
  TxTPlant_Clock_and_time_recording_system_sObjectName                   :T_BA_StateText:='CTR';
  TxTPlant_Clock_and_time_recording_system_sDescription                   :T_BA_StateText:='Clock and time recording system';
// 454 Electro-acoustic systems
  TxTPlant_Electro_acoustic_sound_systems_sObjectName                    :T_BA_StateText:='ELA';
  TxTPlant_Electro_acoustic_sound_systems_sDescription                    :T_BA_StateText:='Electro-acoustic system, sound systems';
  TxTPlant_Conference_and_interpreting_equipment_sObjectName             :T_BA_StateText:='CIE';
  TxTPlant_Conference_and_interpreting_equipment_sDescription             :T_BA_StateText:='Conference and interpreting equipment';
  TxTPlant_Intercom_system_sObjectName                                   :T_BA_StateText:='ICS';
  TxTPlant_Intercom_system_sDescription                                   :T_BA_StateText:='Intercom system';
  TxTPlant_Voice_alarm_system_sObjectName                                :T_BA_StateText:='VAS';
  TxTPlant_Voice_alarm_system_sDescription                                :T_BA_StateText:='Voice alarm system';
  TxTPlant_Intercommunication_systems_sObjectName                        :T_BA_StateText:='ICS';
  TxTPlant_Intercommunication_systems_sDescription                        :T_BA_StateText:='Intercommunication systems';
// 455 Television and antenna systems
  TxTPlant_Television_system_sObjectName                                 :T_BA_StateText:='TVS';
  TxTPlant_Television_system_sDescription                                 :T_BA_StateText:='Television system';
  TxTPlant_Transmitting_and_receiving_antenna_system_sObjectName         :T_BA_StateText:='TRA';
  TxTPlant_Transmitting_and_receiving_antenna_system_sDescription         :T_BA_StateText:='Transmit. and receiving antenna system';
  TxTPlant_BOS_radio_system_sObjectName                                  :T_BA_StateText:='BOS';
  TxTPlant_BOS_radio_system_sDescription                                  :T_BA_StateText:='BOS radio system';
// 456 Hazard detection and alarm systems
  TxTPlant_Fire_detection_and_alarm_system_sObjectName                   :T_BA_StateText:='FDA';
  TxTPlant_Fire_detection_and_alarm_system_sDescription                   :T_BA_StateText:='Fire detection and alarm system';
  TxTPlant_Carbon_monoxide_warning_system_sObjectName                    :T_BA_StateText:='CMW';
  TxTPlant_Carbon_monoxide_warning_system_sDescription                    :T_BA_StateText:='Carbon monoxide warning system';
  TxTPlant_Burglar_alarm_system_sObjectName                              :T_BA_StateText:='BAS';
  TxTPlant_Burglar_alarm_system_sDescription                              :T_BA_StateText:='Burglar alarm system';
  TxTPlant_Fire_control_panel_sObjectName                                :T_BA_StateText:='FCP';
  TxTPlant_Fire_control_panel_sDescription                                :T_BA_StateText:='Fire control panel';
  TxTPlant_Escape_route_protection_system_sObjectName                    :T_BA_StateText:='ERP';
  TxTPlant_Escape_route_protection_system_sDescription                    :T_BA_StateText:='Escape route protection system';
  TxTPlant_Hazard_detection_system_sObjectName                           :T_BA_StateText:='HDS';
  TxTPlant_Hazard_detection_system_sDescription                           :T_BA_StateText:='Hazard detection system';
  TxTPlant_Gas_warning_system_sObjectName                                :T_BA_StateText:='GWS';
  TxTPlant_Gas_warning_system_sDescription                                :T_BA_StateText:='Gas warning system';
  TxTPlant_Smoke_aspiration_system_sObjectName                           :T_BA_StateText:='SAS';
  TxTPlant_Smoke_aspiration_system_sDescription                           :T_BA_StateText:='Smoke aspiration system';
  TxTPlant_Room_observation_system_sObjectName                           :T_BA_StateText:='ROS';
  TxTPlant_Room_observation_system_sDescription                           :T_BA_StateText:='Room observation system';
  TxTPlant_Robbery_alarm_system_sObjectName                              :T_BA_StateText:='ROA';
  TxTPlant_Robbery_alarm_system_sDescription                              :T_BA_StateText:='Robbery alarm system';
  TxTPlant_Guard_control_system_sObjectName                              :T_BA_StateText:='GCS';
  TxTPlant_Guard_control_system_sDescription                              :T_BA_StateText:='Guard control system';
  TxTPlant_Emergency_call_system_sObjectName                             :T_BA_StateText:='EMG';
  TxTPlant_Emergency_call_system_sDescription                             :T_BA_StateText:='Emergency call system';
  TxTPlant_Access_control_system_sObjectName                             :T_BA_StateText:='ACS';
  TxTPlant_Access_control_system_sDescription                             :T_BA_StateText:='Access control system';
// 457 Transmission grids
  TxTPlant_Networks_for_the_transmission_voice_text_etc_sObjectName      :T_BA_StateText:='LAN';
  TxTPlant_Networks_for_the_transmission_voice_text_etc_sDescription      :T_BA_StateText:='Networks  data, voice, text etc';
// 459 Telecommunication and information technology equipment, other
  TxTPlant_Remote_control_systems_sObjectName                            :T_BA_StateText:='RCS';
  TxTPlant_Remote_control_systems_sDescription                            :T_BA_StateText:='Remote control systems';
  TxTPlant_Parking_guidance_systems_sObjectName                          :T_BA_StateText:='PGS';
  TxTPlant_Parking_guidance_systems_sDescription                          :T_BA_StateText:='Parking guidance systems';
// 460 Conveyors
  TxTPlant_File_transportation_systems_sObjectName                       :T_BA_StateText:='FTS';
  TxTPlant_File_transportation_systems_sDescription                       :T_BA_StateText:='File transportation systems';
  TxTPlant_Lift_sObjectName                                              :T_BA_StateText:='LIF';
  TxTPlant_Lift_sDescription                                              :T_BA_StateText:='Lift';
  TxTPlant_Inspection_systems_sObjectName                                :T_BA_StateText:='ISS';
  TxTPlant_Inspection_systems_sDescription                                :T_BA_StateText:='Inspection systems';
  TxTPlant_Moving_walkways_sObjectName                                   :T_BA_StateText:='MWW';
  TxTPlant_Moving_walkways_sDescription                                   :T_BA_StateText:='Moving walkways';
  TxTPlant_Escalators_sObjectName                                        :T_BA_StateText:='ESC';
  TxTPlant_Escalators_sDescription                                        :T_BA_StateText:='Escalators';
  TxTPlant_External_lifts_sObjectName                                    :T_BA_StateText:='EXL';
  TxTPlant_External_lifts_sDescription                                    :T_BA_StateText:='External lifts';
  TxTPlant_Baggage_conveyor_system_sObjectName                           :T_BA_StateText:='BCS';
  TxTPlant_Baggage_conveyor_system_sDescription                           :T_BA_StateText:='Baggage conveyor system';
  TxTPlant_Pneumatic_delivery_systems_sObjectName                        :T_BA_StateText:='PDS';
  TxTPlant_Pneumatic_delivery_systems_sDescription                        :T_BA_StateText:='Pneumatic delivery systems';
  TxTPlant_Goods_transportation_facilities_sObjectName                   :T_BA_StateText:='GTF';
  TxTPlant_Goods_transportation_facilities_sDescription                   :T_BA_StateText:='Goods transportation facilities';
// 470 User-specific systems
// 471 Kitchen technology systems
  TxTPlant_Small_refrigeration_unit_sObjectName                          :T_BA_StateText:='SRU';
  TxTPlant_Small_refrigeration_unit_sDescription                          :T_BA_StateText:='Small refrigeration unit';
// 472 Laundry and cleaning systems
  TxTPlant_Disinfection_unit_sObjectName                                 :T_BA_StateText:='DIS';
  TxTPlant_Disinfection_unit_sDescription                                 :T_BA_StateText:='Disinfection unit';
  TxTPlant_Cleaning_unit_sObjectName                                     :T_BA_StateText:='CLU';
  TxTPlant_Cleaning_unit_sDescription                                     :T_BA_StateText:='Cleaning unit';
  TxTPlant_Sterilisation_systems_sObjectName                             :T_BA_StateText:='STR';
  TxTPlant_Sterilisation_systems_sDescription                             :T_BA_StateText:='Sterilisation systems';
  TxTPlant_Water_treatment_system_sObjectName                            :T_BA_StateText:='WTS';
  TxTPlant_Water_treatment_system_sDescription                            :T_BA_StateText:='Water treatment system';
  TxTPlant_Laundry_system_sObjectName                                    :T_BA_StateText:='LAU';
  TxTPlant_Laundry_system_sDescription                                    :T_BA_StateText:='Laundry system';
// 473 Media supply systems
  TxTPlant_Compressed_air_supply_system_sObjectName                      :T_BA_StateText:='COA';
  TxTPlant_Compressed_air_supply_system_sDescription                      :T_BA_StateText:='Compressed air supply system';
  TxTPlant_Pressure_regulator_unit_sObjectName                           :T_BA_StateText:='PRU';
  TxTPlant_Pressure_regulator_unit_sDescription                           :T_BA_StateText:='Pressure regulator unit';
  TxTPlant_Media_supply_system_sObjectName                               :T_BA_StateText:='MSS';
  TxTPlant_Media_supply_system_sDescription                               :T_BA_StateText:='Media supply system';
  TxTPlant_Medical_and_technical_gases_sObjectName                       :T_BA_StateText:='MTG';
  TxTPlant_Medical_and_technical_gases_sDescription                       :T_BA_StateText:='Medical and technical gases';
  TxTPlant_Vacuum_unit_sObjectName                                       :T_BA_StateText:='VAC';
  TxTPlant_Vacuum_unit_sDescription                                       :T_BA_StateText:='Vacuum unit';
// 474 Medical and laboratory equipment
  TxTPlant_Medical_technical_plant_sObjectName                           :T_BA_StateText:='MED';
  TxTPlant_Medical_technical_plant_sDescription                           :T_BA_StateText:='Medical technical plant';
  TxTPlant_Medical_gas_supply_sObjectName                                :T_BA_StateText:='MGS';
  TxTPlant_Medical_gas_supply_sDescription                                :T_BA_StateText:='Medical gas supply';
  TxTPlant_Laboratory_equipment_sObjectName                              :T_BA_StateText:='LAB';
  TxTPlant_Laboratory_equipment_sDescription                              :T_BA_StateText:='Laboratory equipment (general)';
// 475 Fire extinguishers
  TxTPlant_Fire_extinguisher_sObjectName                                 :T_BA_StateText:='FEG';
  TxTPlant_Fire_extinguisher_sDescription                                 :T_BA_StateText:='Fire extinguisher';
  TxTPlant_Gas_extinguishing_system_sObjectName                          :T_BA_StateText:='GES';
  TxTPlant_Gas_extinguishing_system_sDescription                          :T_BA_StateText:='Gas extinguishing system';
  TxTPlant_Fire_extinguishing_system_sObjectName                         :T_BA_StateText:='FES';
  TxTPlant_Fire_extinguishing_system_sDescription                         :T_BA_StateText:='Fire extinguishing system (general)';
  TxTPlant_Mist_extinguishing_system_sObjectName                         :T_BA_StateText:='MES';
  TxTPlant_Mist_extinguishing_system_sDescription                         :T_BA_StateText:='Mist-extinguishing system';
  TxTPlant_NOX_system_sObjectName                                        :T_BA_StateText:='NOX';
  TxTPlant_NOX_system_sDescription                                        :T_BA_StateText:='NOX system';
  TxTPlant_Sprinkler_system_sObjectName                                  :T_BA_StateText:='SPR';
  TxTPlant_Sprinkler_system_sDescription                                  :T_BA_StateText:='Sprinkler system';
  TxTPlant_Wall_hydrant_system_sObjectName                               :T_BA_StateText:='WHS';
  TxTPlant_Wall_hydrant_system_sDescription                               :T_BA_StateText:='Wall hydrant system';
// 478 Disposal facilities
  TxTPlant_Waste_disposal_system_sObjectName                             :T_BA_StateText:='WDS';
  TxTPlant_Waste_disposal_system_sDescription                             :T_BA_StateText:='Waste disposal system';
  TxTPlant_Media_disposal_system_sObjectName                             :T_BA_StateText:='MDS';
  TxTPlant_Media_disposal_system_sDescription                             :T_BA_StateText:='Media disposal system';
  TxTPlant_Vacuum_cleaning_systems_sObjectName                           :T_BA_StateText:='VCS';
  TxTPlant_Vacuum_cleaning_systems_sDescription                           :T_BA_StateText:='Vacuum cleaning systems';
// 480 Building automation and control systems
  TxTPlant_Automation_control_equipment_sObjectName                      :T_BA_StateText:='ACE';
  TxTPlant_Automation_control_equipment_sDescription                      :T_BA_StateText:='Automation and control equipment';
  TxTPlant_Weather_station_sObjectName                                   :T_BA_StateText:='WET';
  TxTPlant_Weather_station_sDescription                                   :T_BA_StateText:='Weather station';
  TxTPlant_Management_and_operating_equipment_sObjectName                :T_BA_StateText:='MOE';
  TxTPlant_Management_and_operating_equipment_sDescription                :T_BA_StateText:='Management and operating equipment';
  TxTPlant_Room_automation_sObjectName                                   :T_BA_StateText:='RAU';
  TxTPlant_Room_automation_sDescription                                   :T_BA_StateText:='Room automation';
  TxTPlant_Room_automation_system_distributor_sObjectName                :T_BA_StateText:='RAS';
  TxTPlant_Room_automation_system_distributor_sDescription                :T_BA_StateText:='Room automation system distributor';
  TxTPlant_Control_cabinet_sObjectName                                   :T_BA_StateText:='CCB';
  TxTPlant_Control_cabinet_sDescription                                   :T_BA_StateText:='Control cabinet';
  TxTPlant_Settings_sObjectName                                          :T_BA_StateText:='SYP';
  TxTPlant_Settings_sDescription                                          :T_BA_StateText:='System parameters';
  TxTPlant_EventGroups_sObjectName                                       :T_BA_StateText:='EVG';
  TxTPlant_EventGroups_sDescription                                       :T_BA_StateText:='Event groups';
  TxTPlant_Global_Building_Data_sObjectName                              :T_BA_StateText:='GBD';
  TxTPlant_Global_Building_Data_sDescription                              :T_BA_StateText:='global building Data';
// 540 Technical equipment in outdoor facilities
  TxTPlant_Rainwater_retention_basin_sObjectName                         :T_BA_StateText:='RRB';
  TxTPlant_Rainwater_retention_basin_sDescription                         :T_BA_StateText:='Rainwater retention basin';
  TxTPlant_Cistern_system_sObjectName                                    :T_BA_StateText:='CIS';
  TxTPlant_Cistern_system_sDescription                                    :T_BA_StateText:='Cistern system';
END_VAR

// ---- Templates/GVLs/Language/English/TxtTrade_EN.TcGVL
{region '#Template'}
	{attribute 'Version' := '5.0.0.0'}
	{attribute 'Tags' := '"LCID": "1031", "Text": "GVL, DPAD, Trades, ObjectName, Description"'}
	{attribute 'Tags' := '"LCID": "1033", "Text": "GVL, DPAD, Trades, ObjectName, Description"'}
	{attribute 'Description' := '"LCID": "1031", "Text": "Textliste Gewerke"'}
	{attribute 'Description' := '"LCID": "1033", "Text": "Text list trades"'}
{endregion}

{attribute 'global_init_slot' := '40510'}
VAR_GLOBAL
  TxtTrade_Doors_gates_windows_sun_protection_sObjectName                :T_BA_StateText:='Doors, gates, windows, sun protection';
  TxtTrade_Doors_gates_windows_sun_protection_sDescription                :T_BA_StateText:='DGW';
  TxtTrade_Sewage_water_and_gas_plants_sObjectName                       :T_BA_StateText:='Sewage, water and gas plants';
  TxtTrade_Sewage_water_and_gas_plants_sDescription                       :T_BA_StateText:='SWG';
  TxtTrade_Heat_supply_systems_sObjectName                               :T_BA_StateText:='Heat supply systems';
  TxtTrade_Heat_supply_systems_sDescription                               :T_BA_StateText:='HTG';
  TxtTrade_Air_conditioning_sObjectName                                  :T_BA_StateText:='Air conditioning';
  TxtTrade_Air_conditioning_sDescription                                  :T_BA_StateText:='AC_';
  TxtTrade_Refrigeration_systems_sObjectName                             :T_BA_StateText:='Refrigeration systems';
  TxtTrade_Refrigeration_systems_sDescription                             :T_BA_StateText:='RFG';
  TxtTrade_High_voltage_systems_sObjectName                              :T_BA_StateText:='High-voltage systems';
  TxtTrade_High_voltage_systems_sDescription                              :T_BA_StateText:='HVS';
  TxtTrade_Telecommunication_and_information_technology_sObjectName      :T_BA_StateText:='Telecom. and information tech. equipment';
  TxtTrade_Telecommunication_and_information_technology_sDescription      :T_BA_StateText:='TIT';
  TxtTrade_Hazard_detection_and_alarm_systems_sObjectName                :T_BA_StateText:='Hazard detection and alarm systems';
  TxtTrade_Hazard_detection_and_alarm_systems_sDescription                :T_BA_StateText:='HDA';
  TxtTrade_Conveyors_sObjectName                                         :T_BA_StateText:='Conveyors';
  TxtTrade_Conveyors_sDescription                                         :T_BA_StateText:='CVY';
  TxtTrade_Kitchen_technology_systems_sObjectName                        :T_BA_StateText:='Kitchen technology systems';
  TxtTrade_Kitchen_technology_systems_sDescription                        :T_BA_StateText:='KTS';
  TxtTrade_Laundry_and_cleaning_systems_sObjectName                      :T_BA_StateText:='Laundry and cleaning systems';
  TxtTrade_Laundry_and_cleaning_systems_sDescription                      :T_BA_StateText:='LCS';
  TxtTrade_Media_supply_systems_sObjectName                              :T_BA_StateText:='Media supply systems';
  TxtTrade_Media_supply_systems_sDescription                              :T_BA_StateText:='MSS';
  TxtTrade_Medical_and_laboratory_equipment_sObjectName                  :T_BA_StateText:='Medical and laboratory equipment';
  TxtTrade_Medical_and_laboratory_equipment_sDescription                  :T_BA_StateText:='MED';
  TxtTrade_Fire_extinguishing_systems_sObjectName                        :T_BA_StateText:='Fire extinguishing systems';
  TxtTrade_Fire_extinguishing_systems_sDescription                        :T_BA_StateText:='FES';
  TxtTrade_Bathing_facilities_sObjectName                                :T_BA_StateText:='Bathing facilities';
  TxtTrade_Bathing_facilities_sDescription                                :T_BA_StateText:='BTF';
  TxtTrade_Process_heating_cooling_and_air_systems_sObjectName           :T_BA_StateText:='Process heating, cooling and air systems';
  TxtTrade_Process_heating_cooling_and_air_systems_sDescription           :T_BA_StateText:='PRO';
  TxtTrade_Waste_disposal_facilities_sObjectName                         :T_BA_StateText:='Waste disposal facilities';
  TxtTrade_Waste_disposal_facilities_sDescription                         :T_BA_StateText:='WDF';
  TxtTrade_Building_automation_and_control_systems_general_sObjectName   :T_BA_StateText:='Building automation  general';
  TxtTrade_Building_automation_and_control_systems_general_sDescription   :T_BA_StateText:='BAG';
  TxtTrade_Automation_focal_point_information_focal_point_sObjectName    :T_BA_StateText:='Automation focal point';
  TxtTrade_Automation_focal_point_information_focal_point_sDescription    :T_BA_StateText:='AFP';
  TxtTrade_Room_automation_sObjectName                                   :T_BA_StateText:='Room automation';
  TxtTrade_Room_automation_sDescription                                   :T_BA_StateText:='ROM';
  TxtTrade_Outdoor_devices_sObjectName                                   :T_BA_StateText:='Outdoor devices';
  TxtTrade_Outdoor_devices_sDescription                                   :T_BA_StateText:='ODD';
END_VAR

// ---- Templates/GVLs/Language/German/LblAggregates_DE.TcGVL
{region '#Template'}
	{attribute 'Version' := '5.2.0.0'}
	{attribute 'Tags' := '"LCID": "1031", "Text": "GVL, AKS, Labels, ObjectName, Description"'}
	{attribute 'Tags' := '"LCID": "1033", "Text": "GVL, DPAD, Labels, ObjectName, Description"'}
	{attribute 'Description' := '"LCID": "1031", "Text": "Anlagenkennzeichnungssystem, Labels Aggregate"'}
	{attribute 'Description' := '"LCID": "1033", "Text": "Data Point Addressing Description, Labels aggregate"'}
{endregion}
	 
